// TIA Portal V19 export
DATA_BLOCK "Mode Select"   // DB3
{ S7_Optimized_Access := 'TRUE' }
// stored: MemoryReserve 100
   VAR
      "RO Auto" : Bool;
      "RO Manual" : Bool;
      "RO Buffer" : Int;
      "RO Standby" : Bool;
      "RO START" : Bool;
      "RO STOP" : Bool;
      "RO AUTO PROCESS" : Int;
      "RO AUTO STOP PROCES" : Int;
      "MFG MODE" : Struct
         AUTO : Bool;
         MANUAL : Bool;
         STANDBY : Bool;
         BUFFER : Int;
         "AUTO PROCESS BUFF" : Int;
         "AUTO PROCES STOP BUTT" : Int;
         START : Bool;
         STOP : Bool;
      END_STRUCT;
      "HPP PUMP  2 SELECTION" : Bool;
      "HPP PUMP  1 SELECTION" : Bool;
      "RO PUMP 2 SELECTION" : Bool;
      "RO PUMP 1 SELECTION" : Bool;
      "RAW PUMP 1 SELECTION" : Bool;
      "RAW PUMP  2 SELECTION" : Bool;
      "HPP PUMP  2 OUTPUT" : Bool;
      "HPP PUMP  1 OUTPUT" : Bool;
      "RO PUMP 2  OUTPUT" : Bool;
      "RO PUMP 1  OUTPUT" : Bool;
      "RAW PUMP 1  OUTPUT" : Bool;
      "RAW PUMP  2  OUTPUT" : Bool;
   END_VAR
BEGIN
END_DATA_BLOCK
